PROGRAM MAIN
VAR
END_VAR

SqlExpert();

END_PROGRAM

(* stored: Version 1.1.0.1
   POU MAIN: Id {f6d867a2-1c94-4f17-9a9c-61135453d138}, SpecialFunc None *)
